Staubli VAL3: isHexadecimal.pgx

program isHexadecimal(string x_sHex, bool& x_bRes)
  local num i
  local bool l_bFound
  local num j
begin

  for i=0 to len(x_sHex)-1
    l_bFound=false
    for j=0 to len(sDec2HexSymbols)-1
      if mid(x_sHex, 1, i)==sDec2HexSymbols[j]
        l_bFound=true
      endIf
    endFor
    //character not found in the hexadecimal symbol's list
    if !l_bFound
      x_bRes=false
      return
    endIf
  endFor

  x_bRes=true

end
